TYPE ST_Active_RFIDs :
STRUCT
	RFID			: INT;
	CH				: BYTE;
END_STRUCT
END_TYPE

(* stored: Version 1.1.0.1, ProductVersion 3.1.4024.12
   DUT ST_Active_RFIDs: Id {ff240788-82a8-45a7-84f7-980e389f893a} *)
